{attribute 'GeneratedUsingTerminal: EL3201-0030-0022'}
{attribute addProperty BoxType "EL3201-0030-0022"}
{attribute addProperty Id "EtcSlaveTerminalBaseRTDAT %I*RTD_4A3944819WcStateAT %I*WcState_9091E0EB2InfoDataAT %I*InfoData_32EB74EA10"}
{attribute addProperty CRC "4154465977"}
{attribute addProperty Size "21"}
TYPE EL3201_F7A01EB9 EXTENDS EtcSlaveTerminalBase :
STRUCT
	{attribute addProperty Name "RTD"}
	RTD : RTD_4A394481;
	{attribute addProperty Name "WcState"}
	WcState : WcState_9091E0EB;
	{attribute addProperty Name "InfoData"}
	InfoData : InfoData_32EB74EA;
END_STRUCT
END_TYPE

(* stored: Version 1.2.0.0, ProductVersion 3.1.4024.9
   DUT EL3201_F7A01EB9: Id {b18c7678-d22d-42cb-9c8d-9e308fd066de} *)
